// TIA Portal V18 export
FUNCTION_BLOCK "AI"   // FB3, LAD
{ S7_Optimized_Access := 'TRUE' }
VERSION : 0.1
// stored: AutoNumber true, IsIECCheckEnabled false, IsRetainMemResEnabled false, MemoryReserve 100, SetENOAutomatically false, UDAEnableTagReadback false
   VAR_INPUT
      RAW_MIN : Int;
      RAW_MAX : Int;
      SCALE_MIN : Real;
      SCALE_MAX : Real;
      INPUT : Int;
   END_VAR
   VAR_OUTPUT
      FAULT : Bool;
      SCALE_OUT : Real;
      HI_ALRAM : Bool;
      LO_ALRAM : Bool;
   END_VAR
   VAR
      AI { S7_SetPoint := 'True'} : "SCALING";
      MAX_VALUE { S7_SetPoint := 'True'} : Int;
   END_VAR
BEGIN

REGION Network 1 (SCL)

   IF #INPUT < -100 OR  #INPUT > 27648 THEN
       #FAULT :=1;
   ELSE
       #FAULT := 0;
   END_IF;
   IF NOT #FAULT THEN
       #AI(RAW_MIN := #RAW_MIN,
           RAW_MAX := #RAW_MAX,
           INPUT := #INPUT,
           SCALE_MIN := #SCALE_MIN,
           SCALE_MAX := #SCALE_MAX,
           SCALE_OUT => #SCALE_OUT);
   ELSE
       #SCALE_OUT := 0.0;

   END_IF;
       IF #INPUT < 0 THEN
           #LO_ALRAM := 1;
       ELSE
           #LO_ALRAM := 0;
       END_IF;
       IF #INPUT>27648 THEN
           #HI_ALRAM := 1;
       ELSE
           #HI_ALRAM := 0;

        END_IF;
END_REGION
END_FUNCTION_BLOCK
